FUNCTION_BLOCK PUBLIC VehicleManager
VAR_INPUT
	VehicleID		: BYTE;
END_VAR
VAR_OUTPUT
END_VAR
VAR
	
    State 			: eMM_VehicleState := eMM_VehicleState.eVehIdle;
	NextState		: eMM_VehicleState := eMM_VehicleState.eVehIdle;
	NextPos			: REAL := MM_CONST.REJECT_ULOAD_POS;
	NextVel			: REAL := 2.0;
	NextAcc			: REAL := 2.0;
	NextStaIndex	: BYTE := MM_CONST.REJECT_ULOAD_STA;
	CurrStaIndex	: BYTE := MM_CONST.REJECT_ULOAD_STA;
	cmdAck			: BOOL := FALSE;
	cmdCmpl			: BOOL := FALSE;
	TriggerMove		: BOOL := FALSE;
END_VAR

CASE State OF 
	eMM_VehicleState.eVehIdle: //Set Next Move Parameters and then trigger move
	IF (TriggerMove) THEN
		NextState := eMM_VehicleState.eVehMoveCmd_Send;
		TriggerMove := FALSE;
	END_IF
		
	eMM_VehicleState.eVehMoveCmd_Send:	
	    Stations.fbMMSendMsg.M_CmdVehToPos(VehicleID:=VehicleID,Flags:=1,Pos:=NextPos,Acc:=NextAcc,Vel:=NextVel);
		cmdAck := FALSE;
		cmdCmpl := FALSE;
		NextState:= eMM_VehicleState.eVehMoveCmd_WaitAccept; 	
	eMM_VehicleState.eVehMoveCmd_WaitAccept:
		IF (cmdAck) THEN                           //handle cases for timed out here
			NextState := eMM_VehicleState.eVehMoveCmd_WaitCompl;	
            cmdAck := FALSE;		
		END_IF		
	eMM_VehicleState.eVehMoveCmd_WaitCompl:
		IF (cmdCmpl) THEN                         // handle cases for timed out here 
			NextState := eMM_VehicleState.eVehMoveCmd_Compl;
            cmdCmpl := FALSE; 		
		END_IF
	
	eMM_VehicleState.eVehMoveCmd_Reject:
	
    eMM_VehicleState.eVehMoveCmd_Compl:
		NextState := eMM_VehicleState.eVehIdle;
		Stations.fbStationManager.NotifyStationNewVehArrival(Pos:= NextPos, StationIndex:= NextStaIndex, VehicleID:= VehicleID);		
		CurrStaIndex := NextStaIndex;
		
	eMM_VehicleState.eVehMoveTimeOut:
	
    eMM_VehicleState.eError:
	ELSE
	;		
END_CASE
State := NextState;

METHOD PUBLIC M_SetNextMoveParams : BOOL
VAR_INPUT
	Pos :REAL;
	Vel :REAL;
	Acc :REAL;
	StationIndex :BYTE;
END_VAR
NextPos := Pos;
NextVel	:= Vel;
NextAcc	:= Acc;
NextStaIndex := StationIndex;
END_METHOD

PROPERTY PUBLIC MoveCmdAccepted : BOOL
SET
cmdAck := MoveCmdAccepted;
END_SET
END_PROPERTY

PROPERTY PUBLIC MoveCmdCmpl : BOOL
SET
cmdCmpl := MoveCmdCmpl;
END_SET
END_PROPERTY

METHOD PUBLIC ResetVehicleManager : BOOL
VAR_INPUT
END_VAR
    State 			 := eMM_VehicleState.eVehIdle;
	NextState		 := eMM_VehicleState.eVehIdle;
	NextPos			 := MM_CONST.REJECT_ULOAD_POS;
	NextVel			 := 2.0;
	NextAcc			 := 2.0;
	NextStaIndex	 := MM_CONST.REJECT_ULOAD_STA;
	CurrStaIndex	 := MM_CONST.REJECT_ULOAD_STA;
	cmdAck			 := FALSE;
	cmdCmpl			 := FALSE;
	TriggerMove		 := FALSE;
END_METHOD

METHOD PUBLIC ResetVehicleManagerState : BOOL
VAR_INPUT
END_VAR
State := eMM_VehicleState.eVehIdle;
NextState := eMM_VehicleState.eVehIdle;
END_METHOD

PROPERTY PUBLIC TriggerVehMov : BOOL
SET
TriggerMove := TriggerVehMov;
END_SET
END_PROPERTY

PROPERTY PUBLIC VehIdle : BOOL
GET
VehIdle := (State=eMM_VehicleState.eVehIdle);
END_GET
SET
State:=eMM_VehicleState.eVehIdle;
END_SET
END_PROPERTY

END_FUNCTION_BLOCK

(* stored: Version 1.1.0.1, ProductVersion 3.1.4020.12
   POU VehicleManager: Id {c5bc16cb-8a55-4ee1-9986-d239b574ac96}, SpecialFunc None
   Method M_SetNextMoveParams: Id {aa3d2106-ddbf-461f-b6ab-4fa8d8c7c8bd}
   Property MoveCmdAccepted: Id {5368d58c-212d-48f0-9779-f2734980aab8}
   Set Set: Id {15a77724-1405-43a3-9ec7-3fc7625d857c}
   Property MoveCmdCmpl: Id {163e373d-83c9-4549-9306-d0cabf18cd23}
   Set Set: Id {ed25463d-fbcd-46d3-ab99-99114ae299e9}
   Method ResetVehicleManager: Id {ede2e95f-cc15-40a2-a700-14bcc1598ff4}
   Method ResetVehicleManagerState: Id {57a1256f-54cc-4910-bcc1-82a0d8783173}
   Property TriggerVehMov: Id {25983d38-9d9d-481b-b816-fba4635e5311}
   Set Set: Id {ee68445b-b589-45e0-a88c-50b95ae03e3f}
   Property VehIdle: Id {1fd305b8-67ce-4118-aa79-c4f1af3fb6e3}
   Get Get: Id {7ca0cbb9-f649-4053-ac40-9b284ee59069}
   Set Set: Id {8d1b95b2-5d59-4246-ada8-4748e93151b4} *)
